//==================================================================================================
//								RJM Maszyny sp. z o.o.
//									04.06.2022
//	Sterowanie elektrozaworem  
// 	v1.0	|| TC v 3.1.4024.22		|| - pierwsza wersja
//==================================================================================================
INTERFACE ITF_Elektozawor

//==================================================================================================
//								RJM Maszyny sp. z o.o.
//									04.06.2022
//	Sterowanie cewkami elektrozaworu 
// 	v1.0	|| TC v 3.1.4024.22		|| - pierwsza wersja
//==================================================================================================
METHOD Steruj : BOOL
VAR_INPUT
	bKierunekWstrone0						: BOOL;
	bKierunekWStroneMax						: BOOL;	
END_VAR
END_METHOD

END_INTERFACE

(* stored: Version 1.1.0.1, ProductVersion 3.1.4024.11
   Itf ITF_Elektozawor: Id {116db2a7-d9bd-4479-813c-923ad7b3d1ea}
   Method Steruj: Id {78174752-1704-4c0d-a263-8a044f153f3a} *)
